PROGRAM Fahrauftrag //IMPLEMENTS TrajectoryControllable
VAR
	//State machine
	sStart : BOOL := TRUE;
	s0,s1,s2,s3,s4,s5,s6,s7,s8,s9,s10,s11,s12: BOOL := FALSE;
	
	//Auftrag:Auftrag;
	RobotStatusGW1:RobotStatusGW1;
	TrajectoryController:TrajectoryController;
	leererAuftrag:Auftrag;
	//Hilfsvariablen vorübergehend
	//wayPointList : ARRAY[0..1] OF RobotPoseSimple;
END_VAR

//vorübergehend
//wayPointList[0].x := 1400;
//wayPointList[1].x := 1800;
//wayPointList[0].y := 1000;
//wayPointList[1].y := 1000;
//wayPointList[1] := {.x := 1,.y := 2};
leererAuftrag.AbholStation := 0;
leererAuftrag.AbholTasche := 0;
leererAuftrag.AblageStation := 0;
leererAuftrag.AblageTasche := 0;
leererAuftrag.Art := '';

//Frage: Setzt GW3 die Variablen zurück?


//Ablauf einer Fahrt:
IF sStart AND NOT s0 THEN
	sStart := 0; s0 := 1;
	//	RückmeldungGW1 Verfügbar
	Var_HAWIno.Feedback := 'Verfuegbar';
END_IF
//	Warten auf Auftrag
IF s0 AND NOT s1 AND .Var_HAWIno.Auftrag.Art = 'Fahrauftrag' THEN
	s0 := 0; s1 := 1;
	//	RückmeldugGW1 Auftrag angenommen setzt
	Var_HAWIno.Feedback := 'Auftrag angenommen';
	//	Bahnplanung
	//trajectoryControllable.setWaypointList := wayPointList;				//----------todo
END_IF

//	RückmeldungGW3 Fahrt abwarten
IF s1 AND NOT s2 AND trajectoryController.yBoDriving THEN
	s1 := 0; s2 := 1;
	//	RückmeldungGW1 Auf Anfahrt setzen
	Var_HAWIno.Feedback := 'Auf Anfahrt';
END_IF

//	RückmeldungGW3 am Ziel abwarten
IF s2 AND NOT s3 AND trajectoryController.yBoArrivedAtDestination THEN
	s2 := 0; s3 := 1;
	//	Greifersteuerung
																		//----------todo
	//	RückmeldungGW1 Teil aufgenommen setzen
	Var_HAWIno.Feedback := 'Teil aufgenommen';
	//	Fahrauftrag zu Lesekopf
	//trajectoryControllable.setWaypointList := wayPointList;				//----------todo
END_IF

//  RückmeldungGW3 Fahrt abwarten
IF s3 AND NOT s4 AND trajectoryController.yBoDriving THEN
	s3 := 0; s4 := 1;
END_IF

//	RückmeldungGW3 am Ziel abwarten
IF s4 AND NOT s5 AND trajectoryController.yBoArrivedAtDestination THEN
	s4 := 0; s5 := 1;
	//	RückmeldungGW1 Abmeldung
	Var_HAWIno.Feedback := 'Abmeldung';
END_IF

//	Warten auf Werkstück ausgelesen
IF s5 AND NOT s6 AND .Var_HAWIno.RFID_Status = 'WerkstueckAusgelesen' THEN
	s5 := 0; s6 := 1;
	.Var_HAWIno.RFID_Status := '';
	//	Bahnplanung
	//trajectoryControllable.setWaypointList := wayPointList;				//----------todo
END_IF

//	RückmeldungGW3 Fahrt abwarten
IF s6 AND NOT s7 AND trajectoryController.yBoDriving THEN
	s6 := 0; s7 := 1;
	//	Rückmeldung Auf Transport
	Var_HAWIno.Feedback := 'Auf Transport';
END_IF

//	RückmeldungGW3 am Ziel abwarten
IF s7 AND NOT s8 AND trajectoryController.yBoArrivedAtDestination THEN
	s7 := 0; s8 := 1;
	//	RückmeldungGW1 Anmeldung
	Var_HAWIno.Feedback := 'Anmeldung';
END_IF

//	Warten auf Werkstück ausgelesen
IF s8 AND NOT s9 AND .Var_HAWIno.RFID_Status = 'WerkstueckAusgelesen' THEN
	s8 := 0; s9 := 1;
	.Var_HAWIno.RFID_Status := '';
	//	Fahrauftrag zur Ablage
	//trajectoryControllable.setWaypointList := wayPointList;				//----------todo
END_IF

//  RückmeldungGW3 Fahrt abwarten
IF s9 AND NOT s10 AND trajectoryController.yBoDriving THEN
	s9 := 0; s10 := 1;
END_IF

//	RückmeldungGW3 am Ziel abwarten
IF s10 AND NOT s11 AND trajectoryController.yBoArrivedAtDestination THEN
	s10 := 0; s11 := 1;
	//	Greifersteuerung
																		//----------todo
	//	RückmeldungGW1 Teil abgelegt
	Var_HAWIno.Feedback := 'Teil abgelegt';
	//	Fahrauftrag zum Parkplatz
	//trajectoryControllable.setWaypointList := wayPointList;				//----------todo
END_IF

//  RückmeldungGW3 Fahrt abwarten
IF s11 AND NOT s12 AND trajectoryController.yBoDriving THEN
	s11 := 0; s12 := 1;
END_IF

//	RückmeldungGW3 am Ziel abwarten
IF s12 AND NOT s0 AND trajectoryController.yBoArrivedAtDestination THEN
	s12 := 0; s0 := 1;
	.Var_HAWIno.Auftrag := leererAuftrag;
	//	RückmeldungGW1 Verfügbar
	Var_HAWIno.Feedback := 'Verfuegbar';
END_IF

END_PROGRAM

(* stored: Version 1.1.0.1, ProductVersion 3.1.4024.11
   POU Fahrauftrag: Id {d11e2ac1-1df3-4b17-bdc0-8c45421bbbdd}, SpecialFunc None *)
